{attribute 'qualified_only'}
VAR_GLOBAL
	

	
END_VAR

(* stored: Version 1.1.0.1, ProductVersion 3.1.4024.6
   GVL GVL_var: Id {dba55c71-a8a8-4ae4-adce-873cc13bd22c} *)
